// Mitsubishi GX Developer project: Autonomous Cocktail Machine   PLC: FX3U

PROGRAM MAIN
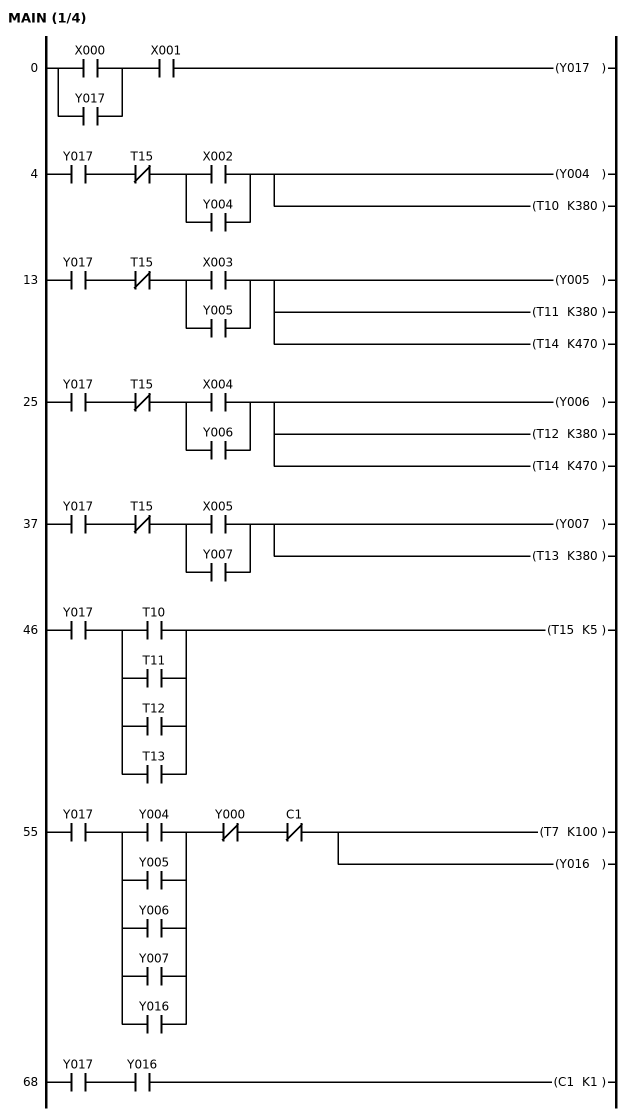
0     LD      X000
      OR      Y017
      AND     X001
      OUT     Y017
4     LD      Y017
      ANI     T15
      LD      X002
      OR      Y004
      ANB
      OUT     Y004
      OUT     T10 K380
13    LD      Y017
      ANI     T15
      LD      X003
      OR      Y005
      ANB
      OUT     Y005
      OUT     T11 K380
      OUT     T14 K470
25    LD      Y017
      ANI     T15
      LD      X004
      OR      Y006
      ANB
      OUT     Y006
      OUT     T12 K380
      OUT     T14 K470
37    LD      Y017
      ANI     T15
      LD      X005
      OR      Y007
      ANB
      OUT     Y007
      OUT     T13 K380
46    LD      Y017
      LD      T10
      OR      T11
      OR      T12
      OR      T13
      ANB
      OUT     T15 K5
55    LD      Y017
      LD      Y004
      OR      Y005
      OR      Y006
      OR      Y007
      OR      Y016
      ANB
      ANI     Y000
      ANI     C1
      OUT     T7 K100
      OUT     Y016
68    LD      Y017
      AND     Y016
      OUT     C1 K1
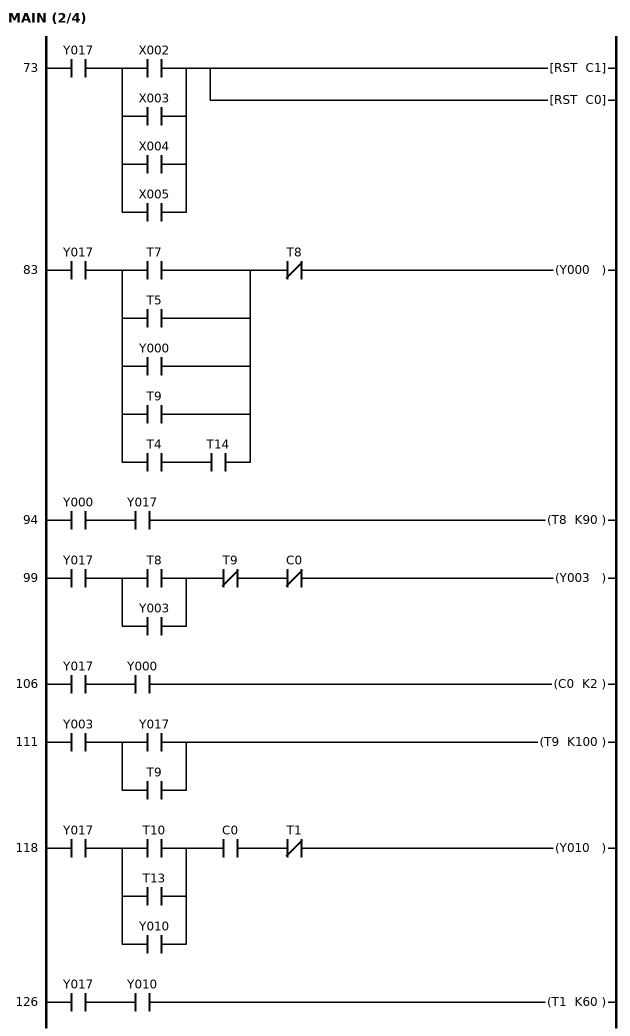
73    LD      Y017
      LD      X002
      OR      X003
      OR      X004
      OR      X005
      ANB
      RST     C1
      RST     C0
83    LD      Y017
      LD      T7
      OR      T5
      OR      Y000
      OR      T9
      LD      T4
      AND     T14
      ORB
      ANB
      ANI     T8
      OUT     Y000
94    LD      Y000
      AND     Y017
      OUT     T8 K90
99    LD      Y017
      LD      T8
      OR      Y003
      ANB
      ANI     T9
      ANI     C0
      OUT     Y003
106   LD      Y017
      AND     Y000
      OUT     C0 K2
111   LD      Y003
      LD      Y017
      OR      T9
      ANB
      OUT     T9 K100
118   LD      Y017
      LD      T10
      OR      T13
      OR      Y010
      ANB
      AND     C0
      ANI     T1
      OUT     Y010
126   LD      Y017
      AND     Y010
      OUT     T1 K60
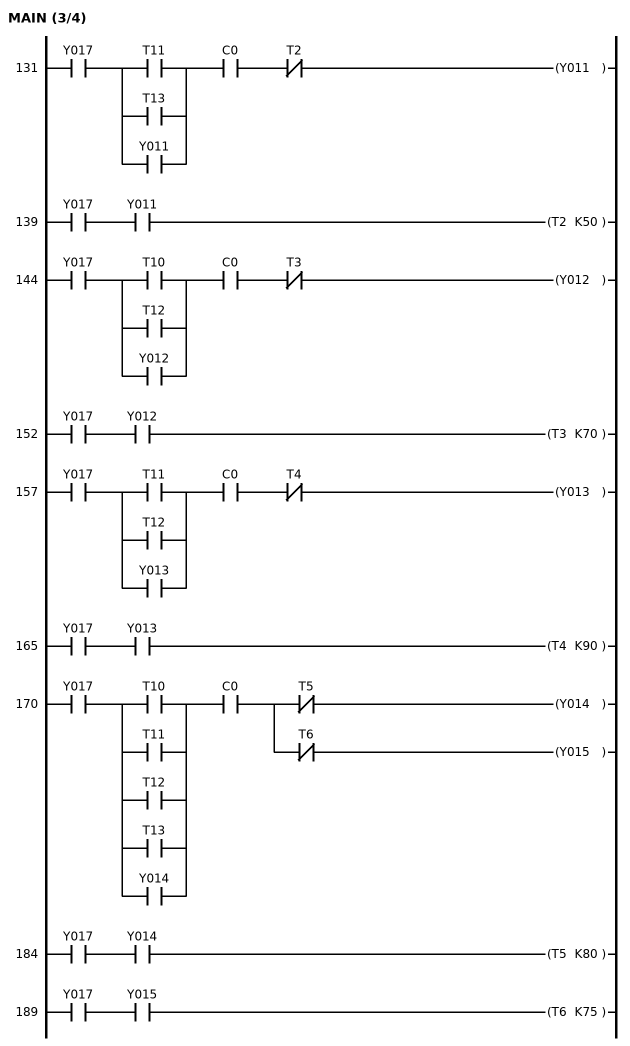
131   LD      Y017
      LD      T11
      OR      T13
      OR      Y011
      ANB
      AND     C0
      ANI     T2
      OUT     Y011
139   LD      Y017
      AND     Y011
      OUT     T2 K50
144   LD      Y017
      LD      T10
      OR      T12
      OR      Y012
      ANB
      AND     C0
      ANI     T3
      OUT     Y012
152   LD      Y017
      AND     Y012
      OUT     T3 K70
157   LD      Y017
      LD      T11
      OR      T12
      OR      Y013
      ANB
      AND     C0
      ANI     T4
      OUT     Y013
165   LD      Y017
      AND     Y013
      OUT     T4 K90
170   LD      Y017
      LD      T10
      OR      T11
      OR      T12
      OR      T13
      OR      Y014
      ANB
      AND     C0
      MPS
      ANI     T5
      OUT     Y014
      MPP
      ANI     T6
      OUT     Y015
184   LD      Y017
      AND     Y014
      OUT     T5 K80
189   LD      Y017
      AND     Y015
      OUT     T6 K75
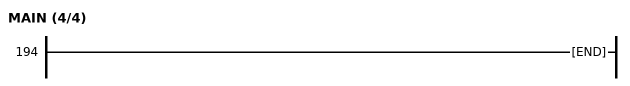
194   END
END_PROGRAM
